FUNCTION_BLOCK ConveyorCTLMulticast (* Basic Function Block Type *)
  (* Standard: 61499-2 *)
  (* Version 0.2, 2003-12-04, JHC, Rockwell Automation, Renamed for better indexing. *)
  (* Version 0.1, 2002-11-05, JHC, Rockwell Automation, Corrected missing ST element in Algorithm REQ. *)
  (* Version 0.0, 2000-05-30, JHC, Rockwell Automation *)
  (* Compiler header: package fb.rt.cs725; *)
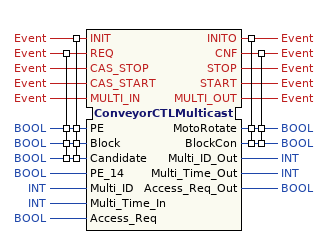
  EVENT_INPUT
    INIT WITH PE, Block, Candidate; (* Initialization Request *)
    REQ WITH PE, Block, Candidate; (* Normal Execution Request *)
    CAS_STOP;
    CAS_START;
    MULTI_IN;
  END_EVENT
  EVENT_OUTPUT
    INITO WITH MotoRotate, BlockCon; (* Initialization Confirm *)
    CNF WITH MotoRotate, BlockCon; (* Execution Confirmation *)
    STOP;
    START;
    MULTI_OUT;
  END_EVENT
  VAR_INPUT
    PE : BOOL; (* Input event qualifier *)
    Block : BOOL;
    Candidate : BOOL;
    PE_14 : BOOL;
    Multi_ID : INT;
    Multi_Time_In : INT;
    Access_Req : BOOL;
  END_VAR
  VAR_OUTPUT
    MotoRotate : BOOL; (* Output event qualifier *)
    BlockCon : BOOL;
    Multi_ID_Out : INT;
    Multi_Time_Out : INT;
    Access_Req_Out : BOOL;
  END_VAR
  VAR
    lastPE : BOOL := 1;
    lastBlock : BOOL := 0;
  END_VAR
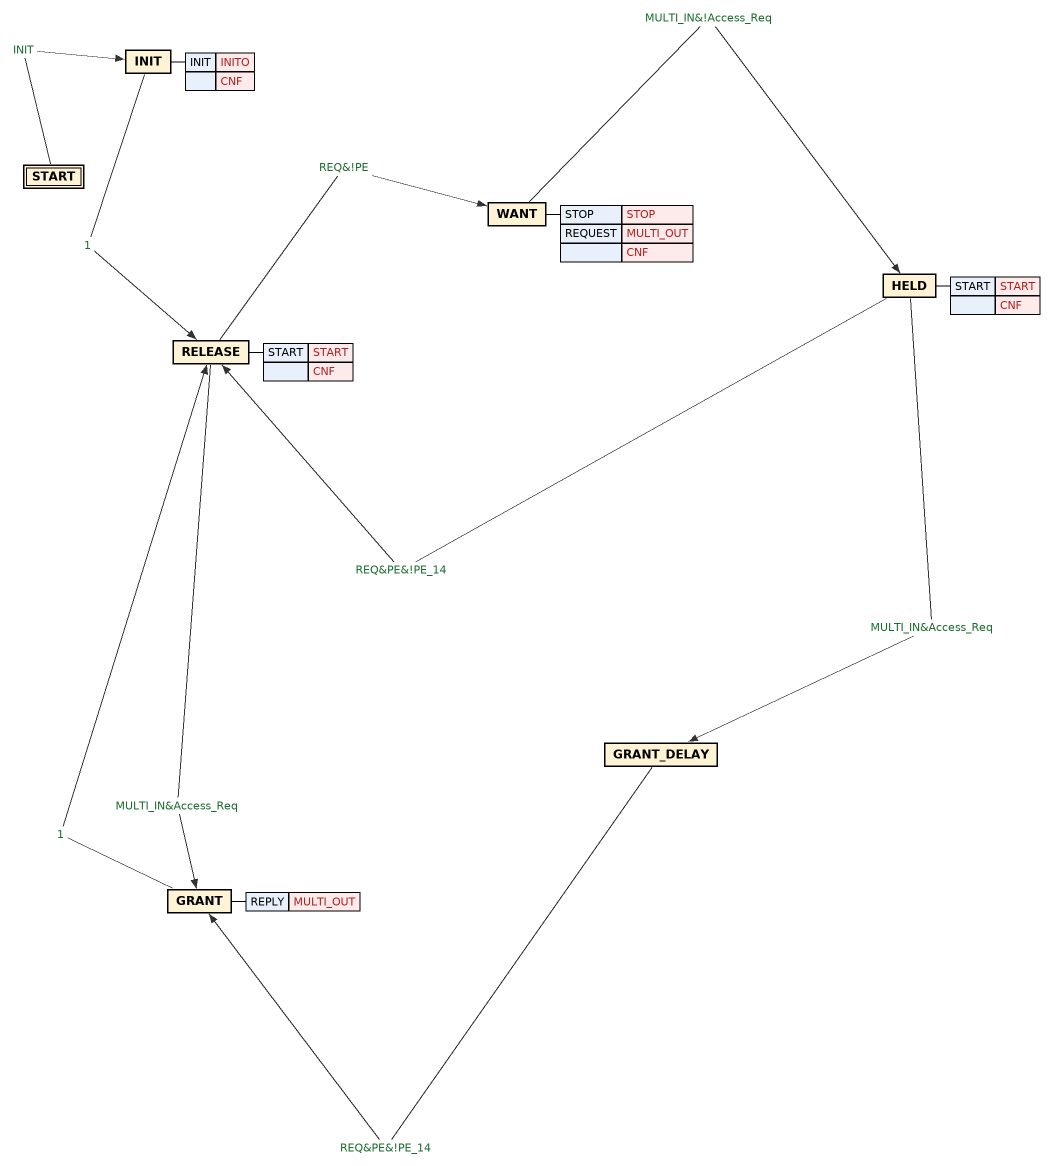
  EC_STATES
    START; (* Initial State *)
    INIT : INIT -> INITO, -> CNF; (* Initialization *)
    RELEASE : START -> START, -> CNF;
    WANT : STOP -> STOP, REQUEST -> MULTI_OUT, -> CNF;
    HELD : START -> START, -> CNF;
    GRANT : REPLY -> MULTI_OUT;
    GRANT_DELAY;
  END_STATES
  EC_TRANSITIONS
    START TO INIT := INIT;
    INIT TO RELEASE := 1;
    RELEASE TO WANT := REQ&!PE;
    WANT TO HELD := MULTI_IN&!Access_Req;
    HELD TO GRANT_DELAY := MULTI_IN&Access_Req;
    GRANT_DELAY TO GRANT := REQ&PE&!PE_14;
    RELEASE TO GRANT := MULTI_IN&Access_Req;
    GRANT TO RELEASE := 1;
    HELD TO RELEASE := REQ&PE&!PE_14;
  END_TRANSITIONS
  ALGORITHM INIT IN ST: (* Initialization algorithm *)
MotoRotate := TRUE;
Block := FALSE;
  END_ALGORITHM
  ALGORITHM REQ IN ST: (* Normally executed algorithm *)
System.out.println(this +  " -> Candidate" + Candidate);
IF Candidate THEN
IF lastPE !:= PE THEN
IF NOT PE THEN
BlockCon:= TRUE;
System.out.println("BlockCon = true");
ELSE
BlockCon:=FALSE;
System.out.println("BlockCon = false");
END_IF
lastPE := PE;
END_IF
IF lastBlock !:= Block THEN
IF Block THEN
STOP.serviceEvent(this);
MotoRotate := FALSE;
System.out.println("Cas Stop");
ELSE
START.serviceEvent(this);
MotoRotate := TRUE;
System.out.println("Cas Start");
END_IF
lastBlock := Block;
END_IF
END_IF
  END_ALGORITHM
  ALGORITHM START IN ST:
MotoRotate:=TRUE;
  END_ALGORITHM
  ALGORITHM STOP IN ST:
MotoRotate := FALSE;
  END_ALGORITHM
  ALGORITHM REQUEST IN Java:
//System.out.println("----------REQUEST----------");
Access_Req_Out.value = true;
  END_ALGORITHM
  ALGORITHM REPLY IN Java:
//System.out.println("----------REPLY----------");
Access_Req_Out.value = false;
  END_ALGORITHM
  ALGORITHM PRINT_GRANT IN Java:
System.out.println(this+"----------GRANT STATE----------");
  END_ALGORITHM
  ALGORITHM PRINT_RELEASED IN Java:
System.out.println(this+"----------RELEASED STATE----------");
  END_ALGORITHM
  ALGORITHM PRINT_WANT IN Java:
System.out.println(this+"----------WANT STATE----------");
  END_ALGORITHM
  ALGORITHM PRINT_HELD IN Java:
System.out.println(this+"----------HELD STATE----------");
  END_ALGORITHM
  ALGORITHM PRINT_TRANSITION IN Java:
System.out.println(this+"----------GRANT DELAY STATE----------");
  END_ALGORITHM
END_FUNCTION_BLOCK
